(* IEC 61131-3 sources: TA/Tests/RetainTest/Man (part 28) *)

(* ---- ManRetainStructureStructureSimple.st ---- *)
PROGRAM ManRetainStructureStructureSimple

IF TRIGGER_IMP.Q AND StartManRetainTest THEN
    RETAINTEST_RETAIN_STRUCTURESTRUCTURESIMPLE.RETAIN.SIMPLE_BOOL := NOT RETAINTEST_RETAIN_STRUCTURESTRUCTURESIMPLE.RETAIN.SIMPLE_BOOL;
    RETAINTEST_RETAIN_STRUCTURESTRUCTURESIMPLE.RETAIN.SIMPLE_BYTE := RETAINTEST_RETAIN_STRUCTURESTRUCTURESIMPLE.RETAIN.SIMPLE_BYTE + 1;
    RETAINTEST_RETAIN_STRUCTURESTRUCTURESIMPLE.RETAIN.SIMPLE_DATE := ANY_TO_DATE(1445385600 + RETAINTEST_RETAIN_STRUCTURESTRUCTURESIMPLE.RETAIN.SIMPLE_DINT * 86400);
    RETAINTEST_RETAIN_STRUCTURESTRUCTURESIMPLE.RETAIN.SIMPLE_DINT := RETAINTEST_RETAIN_STRUCTURESTRUCTURESIMPLE.RETAIN.SIMPLE_DINT + 1;
    RETAINTEST_RETAIN_STRUCTURESTRUCTURESIMPLE.RETAIN.SIMPLE_DWORD := RETAINTEST_RETAIN_STRUCTURESTRUCTURESIMPLE.RETAIN.SIMPLE_DWORD + 1;
    RETAINTEST_RETAIN_STRUCTURESTRUCTURESIMPLE.RETAIN.SIMPLE_INT := RETAINTEST_RETAIN_STRUCTURESTRUCTURESIMPLE.RETAIN.SIMPLE_INT + 1;
    RETAINTEST_RETAIN_STRUCTURESTRUCTURESIMPLE.RETAIN.SIMPLE_LINT := RETAINTEST_RETAIN_STRUCTURESTRUCTURESIMPLE.RETAIN.SIMPLE_LINT + 1;
    RETAINTEST_RETAIN_STRUCTURESTRUCTURESIMPLE.RETAIN.SIMPLE_LREAL := RETAINTEST_RETAIN_STRUCTURESTRUCTURESIMPLE.RETAIN.SIMPLE_LREAL + 1.1;
    RETAINTEST_RETAIN_STRUCTURESTRUCTURESIMPLE.RETAIN.SIMPLE_LWORD := RETAINTEST_RETAIN_STRUCTURESTRUCTURESIMPLE.RETAIN.SIMPLE_LWORD + 1;
    RETAINTEST_RETAIN_STRUCTURESTRUCTURESIMPLE.RETAIN.SIMPLE_REAL := RETAINTEST_RETAIN_STRUCTURESTRUCTURESIMPLE.RETAIN.SIMPLE_REAL + 1.1;
    RETAINTEST_RETAIN_STRUCTURESTRUCTURESIMPLE.RETAIN.SIMPLE_SINT := RETAINTEST_RETAIN_STRUCTURESTRUCTURESIMPLE.RETAIN.SIMPLE_SINT + 1;
    RETAINTEST_RETAIN_STRUCTURESTRUCTURESIMPLE.RETAIN.SIMPLE_STRING := ANY_TO_STRING(RETAINTEST_RETAIN_STRUCTURESTRUCTURESIMPLE.RETAIN.SIMPLE_DINT) + ' ' + ANY_TO_STRING(RETAINTEST_RETAIN_STRUCTURESTRUCTURESIMPLE.RETAIN.SIMPLE_TIME);
    RETAINTEST_RETAIN_STRUCTURESTRUCTURESIMPLE.RETAIN.SIMPLE_TIME := RETAINTEST_RETAIN_STRUCTURESTRUCTURESIMPLE.RETAIN.SIMPLE_TIME + PULSE_TIME;
    RETAINTEST_RETAIN_STRUCTURESTRUCTURESIMPLE.RETAIN.SIMPLE_UDINT := RETAINTEST_RETAIN_STRUCTURESTRUCTURESIMPLE.RETAIN.SIMPLE_UDINT + 1;
    RETAINTEST_RETAIN_STRUCTURESTRUCTURESIMPLE.RETAIN.SIMPLE_UINT := RETAINTEST_RETAIN_STRUCTURESTRUCTURESIMPLE.RETAIN.SIMPLE_UINT + 1;
    RETAINTEST_RETAIN_STRUCTURESTRUCTURESIMPLE.RETAIN.SIMPLE_ULINT := RETAINTEST_RETAIN_STRUCTURESTRUCTURESIMPLE.RETAIN.SIMPLE_ULINT + 1;
    RETAINTEST_RETAIN_STRUCTURESTRUCTURESIMPLE.RETAIN.SIMPLE_USINT := RETAINTEST_RETAIN_STRUCTURESTRUCTURESIMPLE.RETAIN.SIMPLE_USINT + 1;
    RETAINTEST_RETAIN_STRUCTURESTRUCTURESIMPLE.RETAIN.SIMPLE_WORD := RETAINTEST_RETAIN_STRUCTURESTRUCTURESIMPLE.RETAIN.SIMPLE_WORD + 1;

    RETAINTEST_RETAIN_STRUCTURESTRUCTURESIMPLE.NONRETAIN.SIMPLE_BOOL := NOT RETAINTEST_RETAIN_STRUCTURESTRUCTURESIMPLE.NONRETAIN.SIMPLE_BOOL;
    RETAINTEST_RETAIN_STRUCTURESTRUCTURESIMPLE.NONRETAIN.SIMPLE_BYTE := RETAINTEST_RETAIN_STRUCTURESTRUCTURESIMPLE.NONRETAIN.SIMPLE_BYTE + 1;
    RETAINTEST_RETAIN_STRUCTURESTRUCTURESIMPLE.NONRETAIN.SIMPLE_DATE := ANY_TO_DATE(1445385600 + RETAINTEST_RETAIN_STRUCTURESTRUCTURESIMPLE.NONRETAIN.SIMPLE_DINT * 86400);
    RETAINTEST_RETAIN_STRUCTURESTRUCTURESIMPLE.NONRETAIN.SIMPLE_DINT := RETAINTEST_RETAIN_STRUCTURESTRUCTURESIMPLE.NONRETAIN.SIMPLE_DINT + 1;
    RETAINTEST_RETAIN_STRUCTURESTRUCTURESIMPLE.NONRETAIN.SIMPLE_DWORD := RETAINTEST_RETAIN_STRUCTURESTRUCTURESIMPLE.NONRETAIN.SIMPLE_DWORD + 1;
    RETAINTEST_RETAIN_STRUCTURESTRUCTURESIMPLE.NONRETAIN.SIMPLE_INT := RETAINTEST_RETAIN_STRUCTURESTRUCTURESIMPLE.NONRETAIN.SIMPLE_INT + 1;
    RETAINTEST_RETAIN_STRUCTURESTRUCTURESIMPLE.NONRETAIN.SIMPLE_LINT := RETAINTEST_RETAIN_STRUCTURESTRUCTURESIMPLE.NONRETAIN.SIMPLE_LINT + 1;
    RETAINTEST_RETAIN_STRUCTURESTRUCTURESIMPLE.NONRETAIN.SIMPLE_LREAL := RETAINTEST_RETAIN_STRUCTURESTRUCTURESIMPLE.NONRETAIN.SIMPLE_LREAL + 1.1;
    RETAINTEST_RETAIN_STRUCTURESTRUCTURESIMPLE.NONRETAIN.SIMPLE_LWORD := RETAINTEST_RETAIN_STRUCTURESTRUCTURESIMPLE.NONRETAIN.SIMPLE_LWORD + 1;
    RETAINTEST_RETAIN_STRUCTURESTRUCTURESIMPLE.NONRETAIN.SIMPLE_REAL := RETAINTEST_RETAIN_STRUCTURESTRUCTURESIMPLE.NONRETAIN.SIMPLE_REAL + 1.1;
    RETAINTEST_RETAIN_STRUCTURESTRUCTURESIMPLE.NONRETAIN.SIMPLE_SINT := RETAINTEST_RETAIN_STRUCTURESTRUCTURESIMPLE.NONRETAIN.SIMPLE_SINT + 1;
    RETAINTEST_RETAIN_STRUCTURESTRUCTURESIMPLE.NONRETAIN.SIMPLE_STRING := ANY_TO_STRING(RETAINTEST_RETAIN_STRUCTURESTRUCTURESIMPLE.NONRETAIN.SIMPLE_DINT) + ' ' + ANY_TO_STRING(RETAINTEST_RETAIN_STRUCTURESTRUCTURESIMPLE.NONRETAIN.SIMPLE_TIME);
    RETAINTEST_RETAIN_STRUCTURESTRUCTURESIMPLE.NONRETAIN.SIMPLE_TIME := RETAINTEST_RETAIN_STRUCTURESTRUCTURESIMPLE.NONRETAIN.SIMPLE_TIME + PULSE_TIME;
    RETAINTEST_RETAIN_STRUCTURESTRUCTURESIMPLE.NONRETAIN.SIMPLE_UDINT := RETAINTEST_RETAIN_STRUCTURESTRUCTURESIMPLE.NONRETAIN.SIMPLE_UDINT + 1;
    RETAINTEST_RETAIN_STRUCTURESTRUCTURESIMPLE.NONRETAIN.SIMPLE_UINT := RETAINTEST_RETAIN_STRUCTURESTRUCTURESIMPLE.NONRETAIN.SIMPLE_UINT + 1;
    RETAINTEST_RETAIN_STRUCTURESTRUCTURESIMPLE.NONRETAIN.SIMPLE_ULINT := RETAINTEST_RETAIN_STRUCTURESTRUCTURESIMPLE.NONRETAIN.SIMPLE_ULINT + 1;
    RETAINTEST_RETAIN_STRUCTURESTRUCTURESIMPLE.NONRETAIN.SIMPLE_USINT := RETAINTEST_RETAIN_STRUCTURESTRUCTURESIMPLE.NONRETAIN.SIMPLE_USINT + 1;
    RETAINTEST_RETAIN_STRUCTURESTRUCTURESIMPLE.NONRETAIN.SIMPLE_WORD := RETAINTEST_RETAIN_STRUCTURESTRUCTURESIMPLE.NONRETAIN.SIMPLE_WORD + 1;

    RETAINTEST_RETAIN_STRUCTURESTRUCTURESIMPLE.AUTO1.SIMPLE_BOOL := NOT RETAINTEST_RETAIN_STRUCTURESTRUCTURESIMPLE.AUTO1.SIMPLE_BOOL;
    RETAINTEST_RETAIN_STRUCTURESTRUCTURESIMPLE.AUTO1.SIMPLE_BYTE := RETAINTEST_RETAIN_STRUCTURESTRUCTURESIMPLE.AUTO1.SIMPLE_BYTE + 1;
    RETAINTEST_RETAIN_STRUCTURESTRUCTURESIMPLE.AUTO1.SIMPLE_DATE := ANY_TO_DATE(1445385600 + RETAINTEST_RETAIN_STRUCTURESTRUCTURESIMPLE.AUTO1.SIMPLE_DINT * 86400);
    RETAINTEST_RETAIN_STRUCTURESTRUCTURESIMPLE.AUTO1.SIMPLE_DINT := RETAINTEST_RETAIN_STRUCTURESTRUCTURESIMPLE.AUTO1.SIMPLE_DINT + 1;
    RETAINTEST_RETAIN_STRUCTURESTRUCTURESIMPLE.AUTO1.SIMPLE_DWORD := RETAINTEST_RETAIN_STRUCTURESTRUCTURESIMPLE.AUTO1.SIMPLE_DWORD + 1;
    RETAINTEST_RETAIN_STRUCTURESTRUCTURESIMPLE.AUTO1.SIMPLE_INT := RETAINTEST_RETAIN_STRUCTURESTRUCTURESIMPLE.AUTO1.SIMPLE_INT + 1;
    RETAINTEST_RETAIN_STRUCTURESTRUCTURESIMPLE.AUTO1.SIMPLE_LINT := RETAINTEST_RETAIN_STRUCTURESTRUCTURESIMPLE.AUTO1.SIMPLE_LINT + 1;
    RETAINTEST_RETAIN_STRUCTURESTRUCTURESIMPLE.AUTO1.SIMPLE_LREAL := RETAINTEST_RETAIN_STRUCTURESTRUCTURESIMPLE.AUTO1.SIMPLE_LREAL + 1.1;
    RETAINTEST_RETAIN_STRUCTURESTRUCTURESIMPLE.AUTO1.SIMPLE_LWORD := RETAINTEST_RETAIN_STRUCTURESTRUCTURESIMPLE.AUTO1.SIMPLE_LWORD + 1;
    RETAINTEST_RETAIN_STRUCTURESTRUCTURESIMPLE.AUTO1.SIMPLE_REAL := RETAINTEST_RETAIN_STRUCTURESTRUCTURESIMPLE.AUTO1.SIMPLE_REAL + 1.1;
    RETAINTEST_RETAIN_STRUCTURESTRUCTURESIMPLE.AUTO1.SIMPLE_SINT := RETAINTEST_RETAIN_STRUCTURESTRUCTURESIMPLE.AUTO1.SIMPLE_SINT + 1;
    RETAINTEST_RETAIN_STRUCTURESTRUCTURESIMPLE.AUTO1.SIMPLE_STRING := ANY_TO_STRING(RETAINTEST_RETAIN_STRUCTURESTRUCTURESIMPLE.AUTO1.SIMPLE_DINT) + ' ' + ANY_TO_STRING(RETAINTEST_RETAIN_STRUCTURESTRUCTURESIMPLE.AUTO1.SIMPLE_TIME);
    RETAINTEST_RETAIN_STRUCTURESTRUCTURESIMPLE.AUTO1.SIMPLE_TIME := RETAINTEST_RETAIN_STRUCTURESTRUCTURESIMPLE.AUTO1.SIMPLE_TIME + PULSE_TIME;
    RETAINTEST_RETAIN_STRUCTURESTRUCTURESIMPLE.AUTO1.SIMPLE_UDINT := RETAINTEST_RETAIN_STRUCTURESTRUCTURESIMPLE.AUTO1.SIMPLE_UDINT + 1;
    RETAINTEST_RETAIN_STRUCTURESTRUCTURESIMPLE.AUTO1.SIMPLE_UINT := RETAINTEST_RETAIN_STRUCTURESTRUCTURESIMPLE.AUTO1.SIMPLE_UINT + 1;
    RETAINTEST_RETAIN_STRUCTURESTRUCTURESIMPLE.AUTO1.SIMPLE_ULINT := RETAINTEST_RETAIN_STRUCTURESTRUCTURESIMPLE.AUTO1.SIMPLE_ULINT + 1;
    RETAINTEST_RETAIN_STRUCTURESTRUCTURESIMPLE.AUTO1.SIMPLE_USINT := RETAINTEST_RETAIN_STRUCTURESTRUCTURESIMPLE.AUTO1.SIMPLE_USINT + 1;
    RETAINTEST_RETAIN_STRUCTURESTRUCTURESIMPLE.AUTO1.SIMPLE_WORD := RETAINTEST_RETAIN_STRUCTURESTRUCTURESIMPLE.AUTO1.SIMPLE_WORD + 1;

    RETAINTEST_RETAIN_STRUCTURESTRUCTURESIMPLE.AUTO2.SIMPLE_BOOL := RETAINTEST_RETAIN_STRUCTURESTRUCTURESIMPLE.AUTO1.SIMPLE_BOOL;
    RETAINTEST_RETAIN_STRUCTURESTRUCTURESIMPLE.AUTO2.SIMPLE_BYTE := RETAINTEST_RETAIN_STRUCTURESTRUCTURESIMPLE.AUTO1.SIMPLE_BYTE;
    RETAINTEST_RETAIN_STRUCTURESTRUCTURESIMPLE.AUTO2.SIMPLE_DATE := RETAINTEST_RETAIN_STRUCTURESTRUCTURESIMPLE.AUTO1.SIMPLE_DATE;
    RETAINTEST_RETAIN_STRUCTURESTRUCTURESIMPLE.AUTO2.SIMPLE_DINT := RETAINTEST_RETAIN_STRUCTURESTRUCTURESIMPLE.AUTO1.SIMPLE_DINT;
    RETAINTEST_RETAIN_STRUCTURESTRUCTURESIMPLE.AUTO2.SIMPLE_DWORD := RETAINTEST_RETAIN_STRUCTURESTRUCTURESIMPLE.AUTO1.SIMPLE_DWORD;
    RETAINTEST_RETAIN_STRUCTURESTRUCTURESIMPLE.AUTO2.SIMPLE_INT := RETAINTEST_RETAIN_STRUCTURESTRUCTURESIMPLE.AUTO1.SIMPLE_INT;
    RETAINTEST_RETAIN_STRUCTURESTRUCTURESIMPLE.AUTO2.SIMPLE_LINT := RETAINTEST_RETAIN_STRUCTURESTRUCTURESIMPLE.AUTO1.SIMPLE_LINT;
    RETAINTEST_RETAIN_STRUCTURESTRUCTURESIMPLE.AUTO2.SIMPLE_LREAL := RETAINTEST_RETAIN_STRUCTURESTRUCTURESIMPLE.AUTO1.SIMPLE_LREAL;
    RETAINTEST_RETAIN_STRUCTURESTRUCTURESIMPLE.AUTO2.SIMPLE_LWORD := RETAINTEST_RETAIN_STRUCTURESTRUCTURESIMPLE.AUTO1.SIMPLE_LWORD;
    RETAINTEST_RETAIN_STRUCTURESTRUCTURESIMPLE.AUTO2.SIMPLE_REAL := RETAINTEST_RETAIN_STRUCTURESTRUCTURESIMPLE.AUTO1.SIMPLE_REAL;
    RETAINTEST_RETAIN_STRUCTURESTRUCTURESIMPLE.AUTO2.SIMPLE_SINT := RETAINTEST_RETAIN_STRUCTURESTRUCTURESIMPLE.AUTO1.SIMPLE_SINT;
    RETAINTEST_RETAIN_STRUCTURESTRUCTURESIMPLE.AUTO2.SIMPLE_STRING := RETAINTEST_RETAIN_STRUCTURESTRUCTURESIMPLE.AUTO1.SIMPLE_STRING;
    RETAINTEST_RETAIN_STRUCTURESTRUCTURESIMPLE.AUTO2.SIMPLE_TIME := RETAINTEST_RETAIN_STRUCTURESTRUCTURESIMPLE.AUTO1.SIMPLE_TIME;
    RETAINTEST_RETAIN_STRUCTURESTRUCTURESIMPLE.AUTO2.SIMPLE_UDINT := RETAINTEST_RETAIN_STRUCTURESTRUCTURESIMPLE.AUTO1.SIMPLE_UDINT;
    RETAINTEST_RETAIN_STRUCTURESTRUCTURESIMPLE.AUTO2.SIMPLE_UINT := RETAINTEST_RETAIN_STRUCTURESTRUCTURESIMPLE.AUTO1.SIMPLE_UINT;
    RETAINTEST_RETAIN_STRUCTURESTRUCTURESIMPLE.AUTO2.SIMPLE_ULINT := RETAINTEST_RETAIN_STRUCTURESTRUCTURESIMPLE.AUTO1.SIMPLE_ULINT;
    RETAINTEST_RETAIN_STRUCTURESTRUCTURESIMPLE.AUTO2.SIMPLE_USINT := RETAINTEST_RETAIN_STRUCTURESTRUCTURESIMPLE.AUTO1.SIMPLE_USINT;
    RETAINTEST_RETAIN_STRUCTURESTRUCTURESIMPLE.AUTO2.SIMPLE_WORD := RETAINTEST_RETAIN_STRUCTURESTRUCTURESIMPLE.AUTO1.SIMPLE_WORD;

    RETAINTEST_NONRETAIN_STRUCTURESTRUCTURESIMPLE.RETAIN.SIMPLE_BOOL := NOT RETAINTEST_NONRETAIN_STRUCTURESTRUCTURESIMPLE.RETAIN.SIMPLE_BOOL;
    RETAINTEST_NONRETAIN_STRUCTURESTRUCTURESIMPLE.RETAIN.SIMPLE_BYTE := RETAINTEST_NONRETAIN_STRUCTURESTRUCTURESIMPLE.RETAIN.SIMPLE_BYTE + 1;
    RETAINTEST_NONRETAIN_STRUCTURESTRUCTURESIMPLE.RETAIN.SIMPLE_DATE := ANY_TO_DATE(1445385600 + RETAINTEST_NONRETAIN_STRUCTURESTRUCTURESIMPLE.RETAIN.SIMPLE_DINT * 86400);
    RETAINTEST_NONRETAIN_STRUCTURESTRUCTURESIMPLE.RETAIN.SIMPLE_DINT := RETAINTEST_NONRETAIN_STRUCTURESTRUCTURESIMPLE.RETAIN.SIMPLE_DINT + 1;
    RETAINTEST_NONRETAIN_STRUCTURESTRUCTURESIMPLE.RETAIN.SIMPLE_DWORD := RETAINTEST_NONRETAIN_STRUCTURESTRUCTURESIMPLE.RETAIN.SIMPLE_DWORD + 1;
    RETAINTEST_NONRETAIN_STRUCTURESTRUCTURESIMPLE.RETAIN.SIMPLE_INT := RETAINTEST_NONRETAIN_STRUCTURESTRUCTURESIMPLE.RETAIN.SIMPLE_INT + 1;
    RETAINTEST_NONRETAIN_STRUCTURESTRUCTURESIMPLE.RETAIN.SIMPLE_LINT := RETAINTEST_NONRETAIN_STRUCTURESTRUCTURESIMPLE.RETAIN.SIMPLE_LINT + 1;
    RETAINTEST_NONRETAIN_STRUCTURESTRUCTURESIMPLE.RETAIN.SIMPLE_LREAL := RETAINTEST_NONRETAIN_STRUCTURESTRUCTURESIMPLE.RETAIN.SIMPLE_LREAL + 1.1;
    RETAINTEST_NONRETAIN_STRUCTURESTRUCTURESIMPLE.RETAIN.SIMPLE_LWORD := RETAINTEST_NONRETAIN_STRUCTURESTRUCTURESIMPLE.RETAIN.SIMPLE_LWORD + 1;
    RETAINTEST_NONRETAIN_STRUCTURESTRUCTURESIMPLE.RETAIN.SIMPLE_REAL := RETAINTEST_NONRETAIN_STRUCTURESTRUCTURESIMPLE.RETAIN.SIMPLE_REAL + 1.1;
    RETAINTEST_NONRETAIN_STRUCTURESTRUCTURESIMPLE.RETAIN.SIMPLE_SINT := RETAINTEST_NONRETAIN_STRUCTURESTRUCTURESIMPLE.RETAIN.SIMPLE_SINT + 1;
    RETAINTEST_NONRETAIN_STRUCTURESTRUCTURESIMPLE.RETAIN.SIMPLE_STRING := ANY_TO_STRING(RETAINTEST_NONRETAIN_STRUCTURESTRUCTURESIMPLE.RETAIN.SIMPLE_DINT) + ' ' + ANY_TO_STRING(RETAINTEST_NONRETAIN_STRUCTURESTRUCTURESIMPLE.RETAIN.SIMPLE_TIME);
    RETAINTEST_NONRETAIN_STRUCTURESTRUCTURESIMPLE.RETAIN.SIMPLE_TIME := RETAINTEST_NONRETAIN_STRUCTURESTRUCTURESIMPLE.RETAIN.SIMPLE_TIME + PULSE_TIME;
    RETAINTEST_NONRETAIN_STRUCTURESTRUCTURESIMPLE.RETAIN.SIMPLE_UDINT := RETAINTEST_NONRETAIN_STRUCTURESTRUCTURESIMPLE.RETAIN.SIMPLE_UDINT + 1;
    RETAINTEST_NONRETAIN_STRUCTURESTRUCTURESIMPLE.RETAIN.SIMPLE_UINT := RETAINTEST_NONRETAIN_STRUCTURESTRUCTURESIMPLE.RETAIN.SIMPLE_UINT + 1;
    RETAINTEST_NONRETAIN_STRUCTURESTRUCTURESIMPLE.RETAIN.SIMPLE_ULINT := RETAINTEST_NONRETAIN_STRUCTURESTRUCTURESIMPLE.RETAIN.SIMPLE_ULINT + 1;
    RETAINTEST_NONRETAIN_STRUCTURESTRUCTURESIMPLE.RETAIN.SIMPLE_USINT := RETAINTEST_NONRETAIN_STRUCTURESTRUCTURESIMPLE.RETAIN.SIMPLE_USINT + 1;
    RETAINTEST_NONRETAIN_STRUCTURESTRUCTURESIMPLE.RETAIN.SIMPLE_WORD := RETAINTEST_NONRETAIN_STRUCTURESTRUCTURESIMPLE.RETAIN.SIMPLE_WORD + 1;

    RETAINTEST_NONRETAIN_STRUCTURESTRUCTURESIMPLE.NONRETAIN.SIMPLE_BOOL := NOT RETAINTEST_NONRETAIN_STRUCTURESTRUCTURESIMPLE.NONRETAIN.SIMPLE_BOOL;
    RETAINTEST_NONRETAIN_STRUCTURESTRUCTURESIMPLE.NONRETAIN.SIMPLE_BYTE := RETAINTEST_NONRETAIN_STRUCTURESTRUCTURESIMPLE.NONRETAIN.SIMPLE_BYTE + 1;
    RETAINTEST_NONRETAIN_STRUCTURESTRUCTURESIMPLE.NONRETAIN.SIMPLE_DATE := ANY_TO_DATE(1445385600 + RETAINTEST_NONRETAIN_STRUCTURESTRUCTURESIMPLE.NONRETAIN.SIMPLE_DINT * 86400);
    RETAINTEST_NONRETAIN_STRUCTURESTRUCTURESIMPLE.NONRETAIN.SIMPLE_DINT := RETAINTEST_NONRETAIN_STRUCTURESTRUCTURESIMPLE.NONRETAIN.SIMPLE_DINT + 1;
    RETAINTEST_NONRETAIN_STRUCTURESTRUCTURESIMPLE.NONRETAIN.SIMPLE_DWORD := RETAINTEST_NONRETAIN_STRUCTURESTRUCTURESIMPLE.NONRETAIN.SIMPLE_DWORD + 1;
    RETAINTEST_NONRETAIN_STRUCTURESTRUCTURESIMPLE.NONRETAIN.SIMPLE_INT := RETAINTEST_NONRETAIN_STRUCTURESTRUCTURESIMPLE.NONRETAIN.SIMPLE_INT + 1;
    RETAINTEST_NONRETAIN_STRUCTURESTRUCTURESIMPLE.NONRETAIN.SIMPLE_LINT := RETAINTEST_NONRETAIN_STRUCTURESTRUCTURESIMPLE.NONRETAIN.SIMPLE_LINT + 1;
    RETAINTEST_NONRETAIN_STRUCTURESTRUCTURESIMPLE.NONRETAIN.SIMPLE_LREAL := RETAINTEST_NONRETAIN_STRUCTURESTRUCTURESIMPLE.NONRETAIN.SIMPLE_LREAL + 1.1;
    RETAINTEST_NONRETAIN_STRUCTURESTRUCTURESIMPLE.NONRETAIN.SIMPLE_LWORD := RETAINTEST_NONRETAIN_STRUCTURESTRUCTURESIMPLE.NONRETAIN.SIMPLE_LWORD + 1;
    RETAINTEST_NONRETAIN_STRUCTURESTRUCTURESIMPLE.NONRETAIN.SIMPLE_REAL := RETAINTEST_NONRETAIN_STRUCTURESTRUCTURESIMPLE.NONRETAIN.SIMPLE_REAL + 1.1;
    RETAINTEST_NONRETAIN_STRUCTURESTRUCTURESIMPLE.NONRETAIN.SIMPLE_SINT := RETAINTEST_NONRETAIN_STRUCTURESTRUCTURESIMPLE.NONRETAIN.SIMPLE_SINT + 1;
    RETAINTEST_NONRETAIN_STRUCTURESTRUCTURESIMPLE.NONRETAIN.SIMPLE_STRING := ANY_TO_STRING(RETAINTEST_NONRETAIN_STRUCTURESTRUCTURESIMPLE.NONRETAIN.SIMPLE_DINT) + ' ' + ANY_TO_STRING(RETAINTEST_NONRETAIN_STRUCTURESTRUCTURESIMPLE.NONRETAIN.SIMPLE_TIME);
    RETAINTEST_NONRETAIN_STRUCTURESTRUCTURESIMPLE.NONRETAIN.SIMPLE_TIME := RETAINTEST_NONRETAIN_STRUCTURESTRUCTURESIMPLE.NONRETAIN.SIMPLE_TIME + PULSE_TIME;
    RETAINTEST_NONRETAIN_STRUCTURESTRUCTURESIMPLE.NONRETAIN.SIMPLE_UDINT := RETAINTEST_NONRETAIN_STRUCTURESTRUCTURESIMPLE.NONRETAIN.SIMPLE_UDINT + 1;
    RETAINTEST_NONRETAIN_STRUCTURESTRUCTURESIMPLE.NONRETAIN.SIMPLE_UINT := RETAINTEST_NONRETAIN_STRUCTURESTRUCTURESIMPLE.NONRETAIN.SIMPLE_UINT + 1;
    RETAINTEST_NONRETAIN_STRUCTURESTRUCTURESIMPLE.NONRETAIN.SIMPLE_ULINT := RETAINTEST_NONRETAIN_STRUCTURESTRUCTURESIMPLE.NONRETAIN.SIMPLE_ULINT + 1;
    RETAINTEST_NONRETAIN_STRUCTURESTRUCTURESIMPLE.NONRETAIN.SIMPLE_USINT := RETAINTEST_NONRETAIN_STRUCTURESTRUCTURESIMPLE.NONRETAIN.SIMPLE_USINT + 1;
    RETAINTEST_NONRETAIN_STRUCTURESTRUCTURESIMPLE.NONRETAIN.SIMPLE_WORD := RETAINTEST_NONRETAIN_STRUCTURESTRUCTURESIMPLE.NONRETAIN.SIMPLE_WORD + 1;

    RETAINTEST_NONRETAIN_STRUCTURESTRUCTURESIMPLE.AUTO1.SIMPLE_BOOL := NOT RETAINTEST_NONRETAIN_STRUCTURESTRUCTURESIMPLE.AUTO1.SIMPLE_BOOL;
    RETAINTEST_NONRETAIN_STRUCTURESTRUCTURESIMPLE.AUTO1.SIMPLE_BYTE := RETAINTEST_NONRETAIN_STRUCTURESTRUCTURESIMPLE.AUTO1.SIMPLE_BYTE + 1;
    RETAINTEST_NONRETAIN_STRUCTURESTRUCTURESIMPLE.AUTO1.SIMPLE_DATE := ANY_TO_DATE(1445385600 + RETAINTEST_NONRETAIN_STRUCTURESTRUCTURESIMPLE.AUTO1.SIMPLE_DINT * 86400);
    RETAINTEST_NONRETAIN_STRUCTURESTRUCTURESIMPLE.AUTO1.SIMPLE_DINT := RETAINTEST_NONRETAIN_STRUCTURESTRUCTURESIMPLE.AUTO1.SIMPLE_DINT + 1;
    RETAINTEST_NONRETAIN_STRUCTURESTRUCTURESIMPLE.AUTO1.SIMPLE_DWORD := RETAINTEST_NONRETAIN_STRUCTURESTRUCTURESIMPLE.AUTO1.SIMPLE_DWORD + 1;
    RETAINTEST_NONRETAIN_STRUCTURESTRUCTURESIMPLE.AUTO1.SIMPLE_INT := RETAINTEST_NONRETAIN_STRUCTURESTRUCTURESIMPLE.AUTO1.SIMPLE_INT + 1;
    RETAINTEST_NONRETAIN_STRUCTURESTRUCTURESIMPLE.AUTO1.SIMPLE_LINT := RETAINTEST_NONRETAIN_STRUCTURESTRUCTURESIMPLE.AUTO1.SIMPLE_LINT + 1;
    RETAINTEST_NONRETAIN_STRUCTURESTRUCTURESIMPLE.AUTO1.SIMPLE_LREAL := RETAINTEST_NONRETAIN_STRUCTURESTRUCTURESIMPLE.AUTO1.SIMPLE_LREAL + 1.1;
    RETAINTEST_NONRETAIN_STRUCTURESTRUCTURESIMPLE.AUTO1.SIMPLE_LWORD := RETAINTEST_NONRETAIN_STRUCTURESTRUCTURESIMPLE.AUTO1.SIMPLE_LWORD + 1;
    RETAINTEST_NONRETAIN_STRUCTURESTRUCTURESIMPLE.AUTO1.SIMPLE_REAL := RETAINTEST_NONRETAIN_STRUCTURESTRUCTURESIMPLE.AUTO1.SIMPLE_REAL + 1.1;
    RETAINTEST_NONRETAIN_STRUCTURESTRUCTURESIMPLE.AUTO1.SIMPLE_SINT := RETAINTEST_NONRETAIN_STRUCTURESTRUCTURESIMPLE.AUTO1.SIMPLE_SINT + 1;
    RETAINTEST_NONRETAIN_STRUCTURESTRUCTURESIMPLE.AUTO1.SIMPLE_STRING := ANY_TO_STRING(RETAINTEST_NONRETAIN_STRUCTURESTRUCTURESIMPLE.AUTO1.SIMPLE_DINT) + ' ' + ANY_TO_STRING(RETAINTEST_NONRETAIN_STRUCTURESTRUCTURESIMPLE.AUTO1.SIMPLE_TIME);
    RETAINTEST_NONRETAIN_STRUCTURESTRUCTURESIMPLE.AUTO1.SIMPLE_TIME := RETAINTEST_NONRETAIN_STRUCTURESTRUCTURESIMPLE.AUTO1.SIMPLE_TIME + PULSE_TIME;
    RETAINTEST_NONRETAIN_STRUCTURESTRUCTURESIMPLE.AUTO1.SIMPLE_UDINT := RETAINTEST_NONRETAIN_STRUCTURESTRUCTURESIMPLE.AUTO1.SIMPLE_UDINT + 1;
    RETAINTEST_NONRETAIN_STRUCTURESTRUCTURESIMPLE.AUTO1.SIMPLE_UINT := RETAINTEST_NONRETAIN_STRUCTURESTRUCTURESIMPLE.AUTO1.SIMPLE_UINT + 1;
    RETAINTEST_NONRETAIN_STRUCTURESTRUCTURESIMPLE.AUTO1.SIMPLE_ULINT := RETAINTEST_NONRETAIN_STRUCTURESTRUCTURESIMPLE.AUTO1.SIMPLE_ULINT + 1;
    RETAINTEST_NONRETAIN_STRUCTURESTRUCTURESIMPLE.AUTO1.SIMPLE_USINT := RETAINTEST_NONRETAIN_STRUCTURESTRUCTURESIMPLE.AUTO1.SIMPLE_USINT + 1;
    RETAINTEST_NONRETAIN_STRUCTURESTRUCTURESIMPLE.AUTO1.SIMPLE_WORD := RETAINTEST_NONRETAIN_STRUCTURESTRUCTURESIMPLE.AUTO1.SIMPLE_WORD + 1;

    RETAINTEST_NONRETAIN_STRUCTURESTRUCTURESIMPLE.AUTO2.SIMPLE_BOOL := RETAINTEST_NONRETAIN_STRUCTURESTRUCTURESIMPLE.AUTO1.SIMPLE_BOOL;
    RETAINTEST_NONRETAIN_STRUCTURESTRUCTURESIMPLE.AUTO2.SIMPLE_BYTE := RETAINTEST_NONRETAIN_STRUCTURESTRUCTURESIMPLE.AUTO1.SIMPLE_BYTE;
    RETAINTEST_NONRETAIN_STRUCTURESTRUCTURESIMPLE.AUTO2.SIMPLE_DATE := RETAINTEST_NONRETAIN_STRUCTURESTRUCTURESIMPLE.AUTO1.SIMPLE_DATE;
    RETAINTEST_NONRETAIN_STRUCTURESTRUCTURESIMPLE.AUTO2.SIMPLE_DINT := RETAINTEST_NONRETAIN_STRUCTURESTRUCTURESIMPLE.AUTO1.SIMPLE_DINT;
    RETAINTEST_NONRETAIN_STRUCTURESTRUCTURESIMPLE.AUTO2.SIMPLE_DWORD := RETAINTEST_NONRETAIN_STRUCTURESTRUCTURESIMPLE.AUTO1.SIMPLE_DWORD;
    RETAINTEST_NONRETAIN_STRUCTURESTRUCTURESIMPLE.AUTO2.SIMPLE_INT := RETAINTEST_NONRETAIN_STRUCTURESTRUCTURESIMPLE.AUTO1.SIMPLE_INT;
    RETAINTEST_NONRETAIN_STRUCTURESTRUCTURESIMPLE.AUTO2.SIMPLE_LINT := RETAINTEST_NONRETAIN_STRUCTURESTRUCTURESIMPLE.AUTO1.SIMPLE_LINT;
    RETAINTEST_NONRETAIN_STRUCTURESTRUCTURESIMPLE.AUTO2.SIMPLE_LREAL := RETAINTEST_NONRETAIN_STRUCTURESTRUCTURESIMPLE.AUTO1.SIMPLE_LREAL;
    RETAINTEST_NONRETAIN_STRUCTURESTRUCTURESIMPLE.AUTO2.SIMPLE_LWORD := RETAINTEST_NONRETAIN_STRUCTURESTRUCTURESIMPLE.AUTO1.SIMPLE_LWORD;
    RETAINTEST_NONRETAIN_STRUCTURESTRUCTURESIMPLE.AUTO2.SIMPLE_REAL := RETAINTEST_NONRETAIN_STRUCTURESTRUCTURESIMPLE.AUTO1.SIMPLE_REAL;
    RETAINTEST_NONRETAIN_STRUCTURESTRUCTURESIMPLE.AUTO2.SIMPLE_SINT := RETAINTEST_NONRETAIN_STRUCTURESTRUCTURESIMPLE.AUTO1.SIMPLE_SINT;
    RETAINTEST_NONRETAIN_STRUCTURESTRUCTURESIMPLE.AUTO2.SIMPLE_STRING := RETAINTEST_NONRETAIN_STRUCTURESTRUCTURESIMPLE.AUTO1.SIMPLE_STRING;
    RETAINTEST_NONRETAIN_STRUCTURESTRUCTURESIMPLE.AUTO2.SIMPLE_TIME := RETAINTEST_NONRETAIN_STRUCTURESTRUCTURESIMPLE.AUTO1.SIMPLE_TIME;
    RETAINTEST_NONRETAIN_STRUCTURESTRUCTURESIMPLE.AUTO2.SIMPLE_UDINT := RETAINTEST_NONRETAIN_STRUCTURESTRUCTURESIMPLE.AUTO1.SIMPLE_UDINT;
    RETAINTEST_NONRETAIN_STRUCTURESTRUCTURESIMPLE.AUTO2.SIMPLE_UINT := RETAINTEST_NONRETAIN_STRUCTURESTRUCTURESIMPLE.AUTO1.SIMPLE_UINT;
    RETAINTEST_NONRETAIN_STRUCTURESTRUCTURESIMPLE.AUTO2.SIMPLE_ULINT := RETAINTEST_NONRETAIN_STRUCTURESTRUCTURESIMPLE.AUTO1.SIMPLE_ULINT;
    RETAINTEST_NONRETAIN_STRUCTURESTRUCTURESIMPLE.AUTO2.SIMPLE_USINT := RETAINTEST_NONRETAIN_STRUCTURESTRUCTURESIMPLE.AUTO1.SIMPLE_USINT;
    RETAINTEST_NONRETAIN_STRUCTURESTRUCTURESIMPLE.AUTO2.SIMPLE_WORD := RETAINTEST_NONRETAIN_STRUCTURESTRUCTURESIMPLE.AUTO1.SIMPLE_WORD;

    RETAINTEST_AUTO_STRUCTURESTRUCTURESIMPLE.RETAIN.SIMPLE_BOOL := NOT RETAINTEST_AUTO_STRUCTURESTRUCTURESIMPLE.RETAIN.SIMPLE_BOOL;
    RETAINTEST_AUTO_STRUCTURESTRUCTURESIMPLE.RETAIN.SIMPLE_BYTE := RETAINTEST_AUTO_STRUCTURESTRUCTURESIMPLE.RETAIN.SIMPLE_BYTE + 1;
    RETAINTEST_AUTO_STRUCTURESTRUCTURESIMPLE.RETAIN.SIMPLE_DATE := ANY_TO_DATE(1445385600 + RETAINTEST_AUTO_STRUCTURESTRUCTURESIMPLE.RETAIN.SIMPLE_DINT * 86400);
    RETAINTEST_AUTO_STRUCTURESTRUCTURESIMPLE.RETAIN.SIMPLE_DINT := RETAINTEST_AUTO_STRUCTURESTRUCTURESIMPLE.RETAIN.SIMPLE_DINT + 1;
    RETAINTEST_AUTO_STRUCTURESTRUCTURESIMPLE.RETAIN.SIMPLE_DWORD := RETAINTEST_AUTO_STRUCTURESTRUCTURESIMPLE.RETAIN.SIMPLE_DWORD + 1;
    RETAINTEST_AUTO_STRUCTURESTRUCTURESIMPLE.RETAIN.SIMPLE_INT := RETAINTEST_AUTO_STRUCTURESTRUCTURESIMPLE.RETAIN.SIMPLE_INT + 1;
    RETAINTEST_AUTO_STRUCTURESTRUCTURESIMPLE.RETAIN.SIMPLE_LINT := RETAINTEST_AUTO_STRUCTURESTRUCTURESIMPLE.RETAIN.SIMPLE_LINT + 1;
    RETAINTEST_AUTO_STRUCTURESTRUCTURESIMPLE.RETAIN.SIMPLE_LREAL := RETAINTEST_AUTO_STRUCTURESTRUCTURESIMPLE.RETAIN.SIMPLE_LREAL + 1.1;
    RETAINTEST_AUTO_STRUCTURESTRUCTURESIMPLE.RETAIN.SIMPLE_LWORD := RETAINTEST_AUTO_STRUCTURESTRUCTURESIMPLE.RETAIN.SIMPLE_LWORD + 1;
    RETAINTEST_AUTO_STRUCTURESTRUCTURESIMPLE.RETAIN.SIMPLE_REAL := RETAINTEST_AUTO_STRUCTURESTRUCTURESIMPLE.RETAIN.SIMPLE_REAL + 1.1;
    RETAINTEST_AUTO_STRUCTURESTRUCTURESIMPLE.RETAIN.SIMPLE_SINT := RETAINTEST_AUTO_STRUCTURESTRUCTURESIMPLE.RETAIN.SIMPLE_SINT + 1;
    RETAINTEST_AUTO_STRUCTURESTRUCTURESIMPLE.RETAIN.SIMPLE_STRING := ANY_TO_STRING(RETAINTEST_AUTO_STRUCTURESTRUCTURESIMPLE.RETAIN.SIMPLE_DINT) + ' ' + ANY_TO_STRING(RETAINTEST_AUTO_STRUCTURESTRUCTURESIMPLE.RETAIN.SIMPLE_TIME);
    RETAINTEST_AUTO_STRUCTURESTRUCTURESIMPLE.RETAIN.SIMPLE_TIME := RETAINTEST_AUTO_STRUCTURESTRUCTURESIMPLE.RETAIN.SIMPLE_TIME + PULSE_TIME;
    RETAINTEST_AUTO_STRUCTURESTRUCTURESIMPLE.RETAIN.SIMPLE_UDINT := RETAINTEST_AUTO_STRUCTURESTRUCTURESIMPLE.RETAIN.SIMPLE_UDINT + 1;
    RETAINTEST_AUTO_STRUCTURESTRUCTURESIMPLE.RETAIN.SIMPLE_UINT := RETAINTEST_AUTO_STRUCTURESTRUCTURESIMPLE.RETAIN.SIMPLE_UINT + 1;
    RETAINTEST_AUTO_STRUCTURESTRUCTURESIMPLE.RETAIN.SIMPLE_ULINT := RETAINTEST_AUTO_STRUCTURESTRUCTURESIMPLE.RETAIN.SIMPLE_ULINT + 1;
    RETAINTEST_AUTO_STRUCTURESTRUCTURESIMPLE.RETAIN.SIMPLE_USINT := RETAINTEST_AUTO_STRUCTURESTRUCTURESIMPLE.RETAIN.SIMPLE_USINT + 1;
    RETAINTEST_AUTO_STRUCTURESTRUCTURESIMPLE.RETAIN.SIMPLE_WORD := RETAINTEST_AUTO_STRUCTURESTRUCTURESIMPLE.RETAIN.SIMPLE_WORD + 1;

    RETAINTEST_AUTO_STRUCTURESTRUCTURESIMPLE.NONRETAIN.SIMPLE_BOOL := NOT RETAINTEST_AUTO_STRUCTURESTRUCTURESIMPLE.NONRETAIN.SIMPLE_BOOL;
    RETAINTEST_AUTO_STRUCTURESTRUCTURESIMPLE.NONRETAIN.SIMPLE_BYTE := RETAINTEST_AUTO_STRUCTURESTRUCTURESIMPLE.NONRETAIN.SIMPLE_BYTE + 1;
    RETAINTEST_AUTO_STRUCTURESTRUCTURESIMPLE.NONRETAIN.SIMPLE_DATE := ANY_TO_DATE(1445385600 + RETAINTEST_AUTO_STRUCTURESTRUCTURESIMPLE.NONRETAIN.SIMPLE_DINT * 86400);
    RETAINTEST_AUTO_STRUCTURESTRUCTURESIMPLE.NONRETAIN.SIMPLE_DINT := RETAINTEST_AUTO_STRUCTURESTRUCTURESIMPLE.NONRETAIN.SIMPLE_DINT + 1;
    RETAINTEST_AUTO_STRUCTURESTRUCTURESIMPLE.NONRETAIN.SIMPLE_DWORD := RETAINTEST_AUTO_STRUCTURESTRUCTURESIMPLE.NONRETAIN.SIMPLE_DWORD + 1;
    RETAINTEST_AUTO_STRUCTURESTRUCTURESIMPLE.NONRETAIN.SIMPLE_INT := RETAINTEST_AUTO_STRUCTURESTRUCTURESIMPLE.NONRETAIN.SIMPLE_INT + 1;
    RETAINTEST_AUTO_STRUCTURESTRUCTURESIMPLE.NONRETAIN.SIMPLE_LINT := RETAINTEST_AUTO_STRUCTURESTRUCTURESIMPLE.NONRETAIN.SIMPLE_LINT + 1;
    RETAINTEST_AUTO_STRUCTURESTRUCTURESIMPLE.NONRETAIN.SIMPLE_LREAL := RETAINTEST_AUTO_STRUCTURESTRUCTURESIMPLE.NONRETAIN.SIMPLE_LREAL + 1.1;
    RETAINTEST_AUTO_STRUCTURESTRUCTURESIMPLE.NONRETAIN.SIMPLE_LWORD := RETAINTEST_AUTO_STRUCTURESTRUCTURESIMPLE.NONRETAIN.SIMPLE_LWORD + 1;
    RETAINTEST_AUTO_STRUCTURESTRUCTURESIMPLE.NONRETAIN.SIMPLE_REAL := RETAINTEST_AUTO_STRUCTURESTRUCTURESIMPLE.NONRETAIN.SIMPLE_REAL + 1.1;
    RETAINTEST_AUTO_STRUCTURESTRUCTURESIMPLE.NONRETAIN.SIMPLE_SINT := RETAINTEST_AUTO_STRUCTURESTRUCTURESIMPLE.NONRETAIN.SIMPLE_SINT + 1;
    RETAINTEST_AUTO_STRUCTURESTRUCTURESIMPLE.NONRETAIN.SIMPLE_STRING := ANY_TO_STRING(RETAINTEST_AUTO_STRUCTURESTRUCTURESIMPLE.NONRETAIN.SIMPLE_DINT) + ' ' + ANY_TO_STRING(RETAINTEST_AUTO_STRUCTURESTRUCTURESIMPLE.NONRETAIN.SIMPLE_TIME);
    RETAINTEST_AUTO_STRUCTURESTRUCTURESIMPLE.NONRETAIN.SIMPLE_TIME := RETAINTEST_AUTO_STRUCTURESTRUCTURESIMPLE.NONRETAIN.SIMPLE_TIME + PULSE_TIME;
    RETAINTEST_AUTO_STRUCTURESTRUCTURESIMPLE.NONRETAIN.SIMPLE_UDINT := RETAINTEST_AUTO_STRUCTURESTRUCTURESIMPLE.NONRETAIN.SIMPLE_UDINT + 1;
    RETAINTEST_AUTO_STRUCTURESTRUCTURESIMPLE.NONRETAIN.SIMPLE_UINT := RETAINTEST_AUTO_STRUCTURESTRUCTURESIMPLE.NONRETAIN.SIMPLE_UINT + 1;
    RETAINTEST_AUTO_STRUCTURESTRUCTURESIMPLE.NONRETAIN.SIMPLE_ULINT := RETAINTEST_AUTO_STRUCTURESTRUCTURESIMPLE.NONRETAIN.SIMPLE_ULINT + 1;
    RETAINTEST_AUTO_STRUCTURESTRUCTURESIMPLE.NONRETAIN.SIMPLE_USINT := RETAINTEST_AUTO_STRUCTURESTRUCTURESIMPLE.NONRETAIN.SIMPLE_USINT + 1;
    RETAINTEST_AUTO_STRUCTURESTRUCTURESIMPLE.NONRETAIN.SIMPLE_WORD := RETAINTEST_AUTO_STRUCTURESTRUCTURESIMPLE.NONRETAIN.SIMPLE_WORD + 1;

    RETAINTEST_AUTO_STRUCTURESTRUCTURESIMPLE.AUTO1.SIMPLE_BOOL := NOT RETAINTEST_AUTO_STRUCTURESTRUCTURESIMPLE.AUTO1.SIMPLE_BOOL;
    RETAINTEST_AUTO_STRUCTURESTRUCTURESIMPLE.AUTO1.SIMPLE_BYTE := RETAINTEST_AUTO_STRUCTURESTRUCTURESIMPLE.AUTO1.SIMPLE_BYTE + 1;
    RETAINTEST_AUTO_STRUCTURESTRUCTURESIMPLE.AUTO1.SIMPLE_DATE := ANY_TO_DATE(1445385600 + RETAINTEST_AUTO_STRUCTURESTRUCTURESIMPLE.AUTO1.SIMPLE_DINT * 86400);
    RETAINTEST_AUTO_STRUCTURESTRUCTURESIMPLE.AUTO1.SIMPLE_DINT := RETAINTEST_AUTO_STRUCTURESTRUCTURESIMPLE.AUTO1.SIMPLE_DINT + 1;
    RETAINTEST_AUTO_STRUCTURESTRUCTURESIMPLE.AUTO1.SIMPLE_DWORD := RETAINTEST_AUTO_STRUCTURESTRUCTURESIMPLE.AUTO1.SIMPLE_DWORD + 1;
    RETAINTEST_AUTO_STRUCTURESTRUCTURESIMPLE.AUTO1.SIMPLE_INT := RETAINTEST_AUTO_STRUCTURESTRUCTURESIMPLE.AUTO1.SIMPLE_INT + 1;
    RETAINTEST_AUTO_STRUCTURESTRUCTURESIMPLE.AUTO1.SIMPLE_LINT := RETAINTEST_AUTO_STRUCTURESTRUCTURESIMPLE.AUTO1.SIMPLE_LINT + 1;
    RETAINTEST_AUTO_STRUCTURESTRUCTURESIMPLE.AUTO1.SIMPLE_LREAL := RETAINTEST_AUTO_STRUCTURESTRUCTURESIMPLE.AUTO1.SIMPLE_LREAL + 1.1;
    RETAINTEST_AUTO_STRUCTURESTRUCTURESIMPLE.AUTO1.SIMPLE_LWORD := RETAINTEST_AUTO_STRUCTURESTRUCTURESIMPLE.AUTO1.SIMPLE_LWORD + 1;
    RETAINTEST_AUTO_STRUCTURESTRUCTURESIMPLE.AUTO1.SIMPLE_REAL := RETAINTEST_AUTO_STRUCTURESTRUCTURESIMPLE.AUTO1.SIMPLE_REAL + 1.1;
    RETAINTEST_AUTO_STRUCTURESTRUCTURESIMPLE.AUTO1.SIMPLE_SINT := RETAINTEST_AUTO_STRUCTURESTRUCTURESIMPLE.AUTO1.SIMPLE_SINT + 1;
    RETAINTEST_AUTO_STRUCTURESTRUCTURESIMPLE.AUTO1.SIMPLE_STRING := ANY_TO_STRING(RETAINTEST_AUTO_STRUCTURESTRUCTURESIMPLE.AUTO1.SIMPLE_DINT) + ' ' + ANY_TO_STRING(RETAINTEST_AUTO_STRUCTURESTRUCTURESIMPLE.AUTO1.SIMPLE_TIME);
    RETAINTEST_AUTO_STRUCTURESTRUCTURESIMPLE.AUTO1.SIMPLE_TIME := RETAINTEST_AUTO_STRUCTURESTRUCTURESIMPLE.AUTO1.SIMPLE_TIME + PULSE_TIME;
    RETAINTEST_AUTO_STRUCTURESTRUCTURESIMPLE.AUTO1.SIMPLE_UDINT := RETAINTEST_AUTO_STRUCTURESTRUCTURESIMPLE.AUTO1.SIMPLE_UDINT + 1;
    RETAINTEST_AUTO_STRUCTURESTRUCTURESIMPLE.AUTO1.SIMPLE_UINT := RETAINTEST_AUTO_STRUCTURESTRUCTURESIMPLE.AUTO1.SIMPLE_UINT + 1;
    RETAINTEST_AUTO_STRUCTURESTRUCTURESIMPLE.AUTO1.SIMPLE_ULINT := RETAINTEST_AUTO_STRUCTURESTRUCTURESIMPLE.AUTO1.SIMPLE_ULINT + 1;
    RETAINTEST_AUTO_STRUCTURESTRUCTURESIMPLE.AUTO1.SIMPLE_USINT := RETAINTEST_AUTO_STRUCTURESTRUCTURESIMPLE.AUTO1.SIMPLE_USINT + 1;
    RETAINTEST_AUTO_STRUCTURESTRUCTURESIMPLE.AUTO1.SIMPLE_WORD := RETAINTEST_AUTO_STRUCTURESTRUCTURESIMPLE.AUTO1.SIMPLE_WORD + 1;

    RETAINTEST_AUTO_STRUCTURESTRUCTURESIMPLE.AUTO2.SIMPLE_BOOL := RETAINTEST_AUTO_STRUCTURESTRUCTURESIMPLE.AUTO1.SIMPLE_BOOL;
    RETAINTEST_AUTO_STRUCTURESTRUCTURESIMPLE.AUTO2.SIMPLE_BYTE := RETAINTEST_AUTO_STRUCTURESTRUCTURESIMPLE.AUTO1.SIMPLE_BYTE;
    RETAINTEST_AUTO_STRUCTURESTRUCTURESIMPLE.AUTO2.SIMPLE_DATE := RETAINTEST_AUTO_STRUCTURESTRUCTURESIMPLE.AUTO1.SIMPLE_DATE;
    RETAINTEST_AUTO_STRUCTURESTRUCTURESIMPLE.AUTO2.SIMPLE_DINT := RETAINTEST_AUTO_STRUCTURESTRUCTURESIMPLE.AUTO1.SIMPLE_DINT;
    RETAINTEST_AUTO_STRUCTURESTRUCTURESIMPLE.AUTO2.SIMPLE_DWORD := RETAINTEST_AUTO_STRUCTURESTRUCTURESIMPLE.AUTO1.SIMPLE_DWORD;
    RETAINTEST_AUTO_STRUCTURESTRUCTURESIMPLE.AUTO2.SIMPLE_INT := RETAINTEST_AUTO_STRUCTURESTRUCTURESIMPLE.AUTO1.SIMPLE_INT;
    RETAINTEST_AUTO_STRUCTURESTRUCTURESIMPLE.AUTO2.SIMPLE_LINT := RETAINTEST_AUTO_STRUCTURESTRUCTURESIMPLE.AUTO1.SIMPLE_LINT;
    RETAINTEST_AUTO_STRUCTURESTRUCTURESIMPLE.AUTO2.SIMPLE_LREAL := RETAINTEST_AUTO_STRUCTURESTRUCTURESIMPLE.AUTO1.SIMPLE_LREAL;
    RETAINTEST_AUTO_STRUCTURESTRUCTURESIMPLE.AUTO2.SIMPLE_LWORD := RETAINTEST_AUTO_STRUCTURESTRUCTURESIMPLE.AUTO1.SIMPLE_LWORD;
    RETAINTEST_AUTO_STRUCTURESTRUCTURESIMPLE.AUTO2.SIMPLE_REAL := RETAINTEST_AUTO_STRUCTURESTRUCTURESIMPLE.AUTO1.SIMPLE_REAL;
    RETAINTEST_AUTO_STRUCTURESTRUCTURESIMPLE.AUTO2.SIMPLE_SINT := RETAINTEST_AUTO_STRUCTURESTRUCTURESIMPLE.AUTO1.SIMPLE_SINT;
    RETAINTEST_AUTO_STRUCTURESTRUCTURESIMPLE.AUTO2.SIMPLE_STRING := RETAINTEST_AUTO_STRUCTURESTRUCTURESIMPLE.AUTO1.SIMPLE_STRING;
    RETAINTEST_AUTO_STRUCTURESTRUCTURESIMPLE.AUTO2.SIMPLE_TIME := RETAINTEST_AUTO_STRUCTURESTRUCTURESIMPLE.AUTO1.SIMPLE_TIME;
    RETAINTEST_AUTO_STRUCTURESTRUCTURESIMPLE.AUTO2.SIMPLE_UDINT := RETAINTEST_AUTO_STRUCTURESTRUCTURESIMPLE.AUTO1.SIMPLE_UDINT;
    RETAINTEST_AUTO_STRUCTURESTRUCTURESIMPLE.AUTO2.SIMPLE_UINT := RETAINTEST_AUTO_STRUCTURESTRUCTURESIMPLE.AUTO1.SIMPLE_UINT;
    RETAINTEST_AUTO_STRUCTURESTRUCTURESIMPLE.AUTO2.SIMPLE_ULINT := RETAINTEST_AUTO_STRUCTURESTRUCTURESIMPLE.AUTO1.SIMPLE_ULINT;
    RETAINTEST_AUTO_STRUCTURESTRUCTURESIMPLE.AUTO2.SIMPLE_USINT := RETAINTEST_AUTO_STRUCTURESTRUCTURESIMPLE.AUTO1.SIMPLE_USINT;
    RETAINTEST_AUTO_STRUCTURESTRUCTURESIMPLE.AUTO2.SIMPLE_WORD := RETAINTEST_AUTO_STRUCTURESTRUCTURESIMPLE.AUTO1.SIMPLE_WORD;
END_IF;

END_PROGRAM
